// LS Electric XG5000 project: 신호등
// PLC LSPLC

PROGRAM 신호등 (task: 스캔 프로그램)

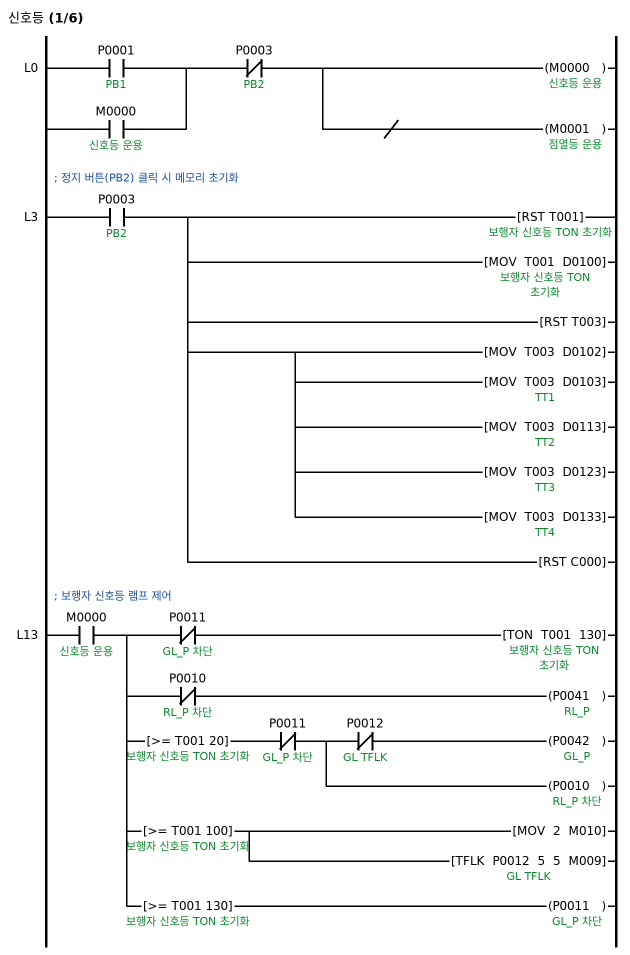
; L0
LOAD      P0001	// PB1
OR        M0000	// 신호등 운용
AND NOT   P0003	// PB2
OUT       M0000	// 신호등 운용
NOT
OUT       M0001	// 점멸등 운용
// 정지 버튼(PB2) 클릭 시 메모리 초기화
; L3
LOAD      P0003	// PB2
RST       T001	// 보행자 신호등 TON 초기화
MOV       T001 D0100	// 보행자 신호등 TON 초기화
RST       T003
MOV       T003 D0102
MOV       T003 D0103	// TT1
MOV       T003 D0113	// TT2
MOV       T003 D0123	// TT3
MOV       T003 D0133	// TT4
RST       C000
// 보행자 신호등 램프 제어
; L13
LOAD      M0000	// 신호등 운용
MPUSH
AND NOT   P0011	// GL_P 차단
TON       T001 130	// 보행자 신호등 TON 초기화
MLOAD
AND NOT   P0010	// RL_P 차단
OUT       P0041	// RL_P
MLOAD
AND>=     T001 20	// 보행자 신호등 TON 초기화
AND NOT   P0011	// GL_P 차단
MPUSH
AND NOT   P0012	// GL TFLK
OUT       P0042	// GL_P
MPOP
OUT       P0010	// RL_P 차단
MLOAD
AND>=     T001 100	// 보행자 신호등 TON 초기화
MOV       2 M010
TFLK      P0012 5 5 M009	// GL TFLK
MPOP
AND>=     T001 130	// 보행자 신호등 TON 초기화
OUT       P0011	// GL_P 차단

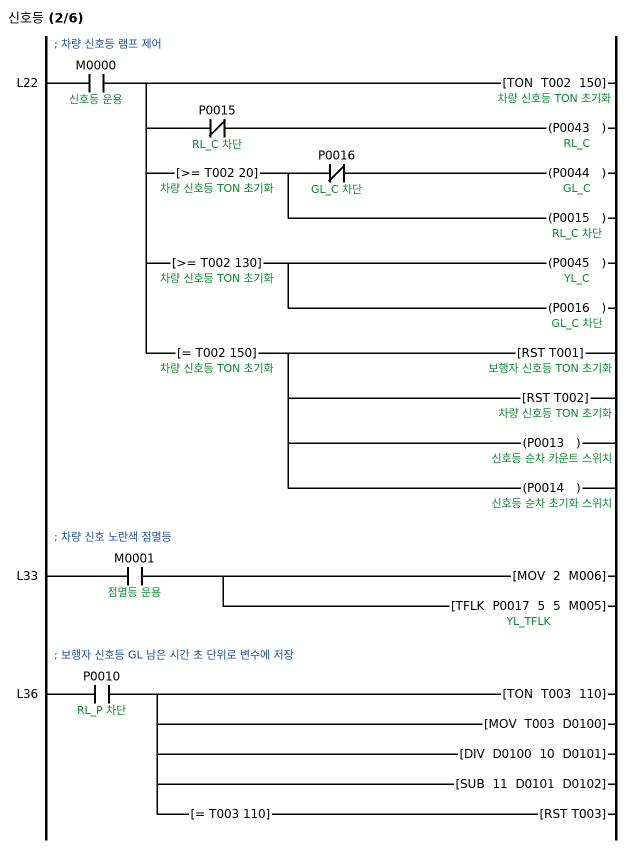
// 차량 신호등 램프 제어
; L22
LOAD      M0000	// 신호등 운용
TON       T002 150	// 차량 신호등 TON 초기화
MPUSH
AND NOT   P0015	// RL_C 차단
OUT       P0043	// RL_C
MLOAD
AND>=     T002 20	// 차량 신호등 TON 초기화
MPUSH
AND NOT   P0016	// GL_C 차단
OUT       P0044	// GL_C
MPOP
OUT       P0015	// RL_C 차단
MLOAD
AND>=     T002 130	// 차량 신호등 TON 초기화
OUT       P0045	// YL_C
OUT       P0016	// GL_C 차단
MPOP
AND=      T002 150	// 차량 신호등 TON 초기화
RST       T001	// 보행자 신호등 TON 초기화
RST       T002	// 차량 신호등 TON 초기화
OUT       P0013	// 신호등 순차 카운트 스위치
OUT       P0014	// 신호등 순차 초기화 스위치
// 차량 신호 노란색 점멸등 
; L33
LOAD      M0001	// 점멸등 운용
MOV       2 M006
TFLK      P0017 5 5 M005	// YL_TFLK
// 보행자 신호등 GL 남은 시간 초 단위로 변수에 저장
; L36
LOAD      P0010	// RL_P 차단
TON       T003 110
MOV       T003 D0100
DIV       D0100 10 D0101
SUB       11 D0101 D0102
AND=      T003 110
RST       T003

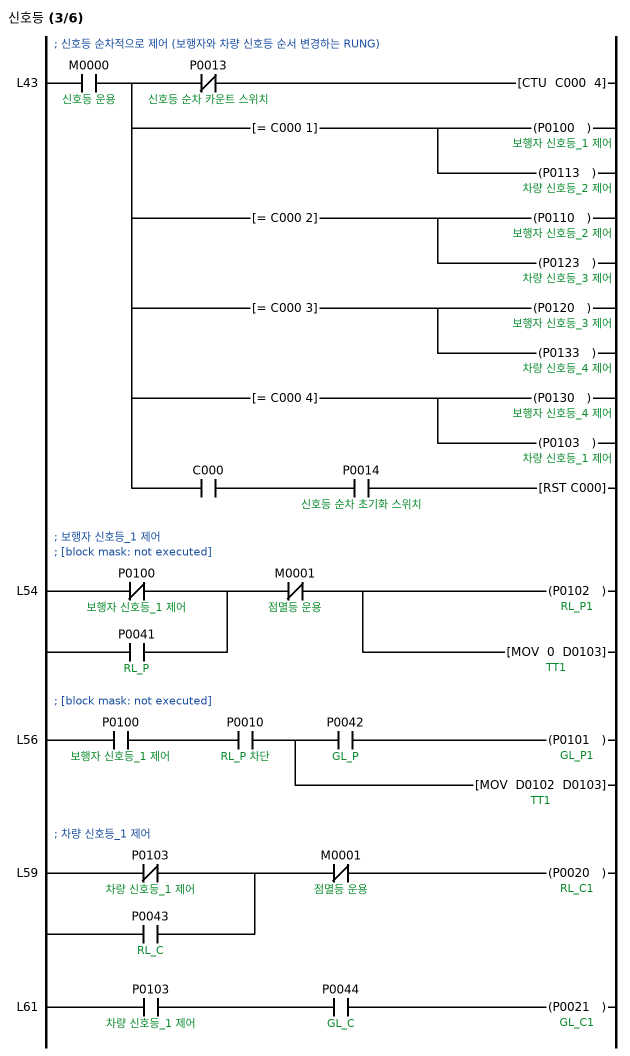
// 신호등 순차적으로 제어 (보행자와 차량 신호등 순서 변경하는 RUNG)
; L43
LOAD      M0000	// 신호등 운용
MPUSH
AND NOT   P0013	// 신호등 순차 카운트 스위치
CTU       C000 4
MLOAD
AND=      C000 1
OUT       P0100	// 보행자 신호등_1 제어
OUT       P0113	// 차량 신호등_2 제어
MLOAD
AND=      C000 2
OUT       P0110	// 보행자 신호등_2 제어
OUT       P0123	// 차량 신호등_3 제어
MLOAD
AND=      C000 3
OUT       P0120	// 보행자 신호등_3 제어
OUT       P0133	// 차량 신호등_4 제어
MLOAD
AND=      C000 4
OUT       P0130	// 보행자 신호등_4 제어
OUT       P0103	// 차량 신호등_1 제어
MPOP
AND       C000
AND       P0014	// 신호등 순차 초기화 스위치
RST       C000
// 보행자 신호등_1 제어
; L54 (block mask: not executed)
LOAD NOT  P0100	// 보행자 신호등_1 제어
OR        P0041	// RL_P
AND NOT   M0001	// 점멸등 운용
OUT       P0102	// RL_P1
MOV       0 D0103	// TT1
; L56 (block mask: not executed)
LOAD      P0100	// 보행자 신호등_1 제어
AND       P0010	// RL_P 차단
MPUSH
AND       P0042	// GL_P
OUT       P0101	// GL_P1
MPOP
MOV       D0102 D0103	// TT1
// 차량 신호등_1 제어
; L59
LOAD NOT  P0103	// 차량 신호등_1 제어
OR        P0043	// RL_C
AND NOT   M0001	// 점멸등 운용
OUT       P0020	// RL_C1
; L61
LOAD      P0103	// 차량 신호등_1 제어
AND       P0044	// GL_C
OUT       P0021	// GL_C1

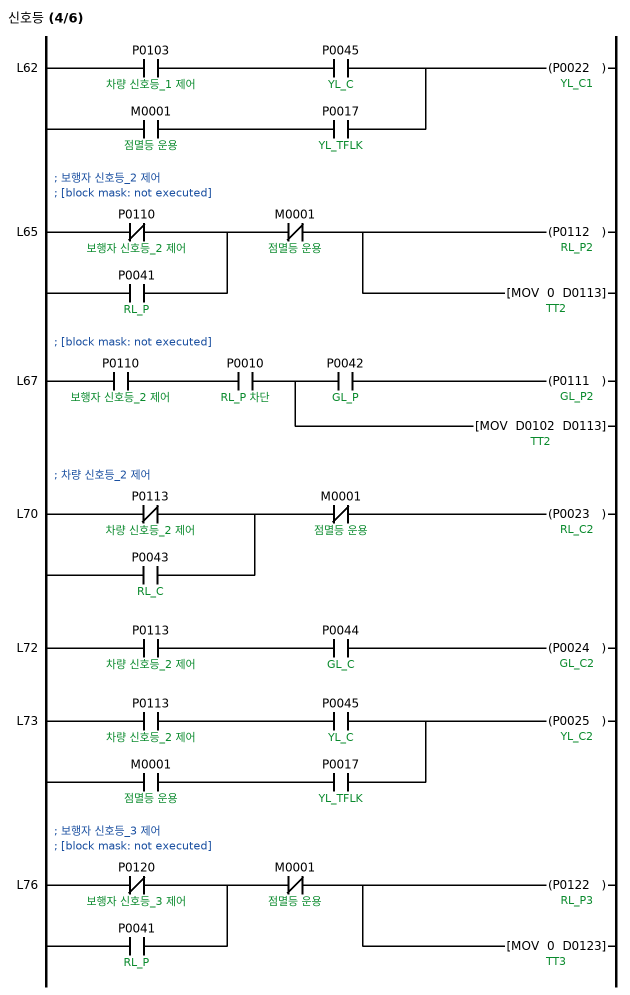
; L62
LOAD      P0103	// 차량 신호등_1 제어
AND       P0045	// YL_C
LOAD      M0001	// 점멸등 운용
AND       P0017	// YL_TFLK
OR LOAD
OUT       P0022	// YL_C1
// 보행자 신호등_2 제어
; L65 (block mask: not executed)
LOAD NOT  P0110	// 보행자 신호등_2 제어
OR        P0041	// RL_P
AND NOT   M0001	// 점멸등 운용
OUT       P0112	// RL_P2
MOV       0 D0113	// TT2
; L67 (block mask: not executed)
LOAD      P0110	// 보행자 신호등_2 제어
AND       P0010	// RL_P 차단
MPUSH
AND       P0042	// GL_P
OUT       P0111	// GL_P2
MPOP
MOV       D0102 D0113	// TT2
// 차량 신호등_2 제어
; L70
LOAD NOT  P0113	// 차량 신호등_2 제어
OR        P0043	// RL_C
AND NOT   M0001	// 점멸등 운용
OUT       P0023	// RL_C2
; L72
LOAD      P0113	// 차량 신호등_2 제어
AND       P0044	// GL_C
OUT       P0024	// GL_C2
; L73
LOAD      P0113	// 차량 신호등_2 제어
AND       P0045	// YL_C
LOAD      M0001	// 점멸등 운용
AND       P0017	// YL_TFLK
OR LOAD
OUT       P0025	// YL_C2
// 보행자 신호등_3 제어
; L76 (block mask: not executed)
LOAD NOT  P0120	// 보행자 신호등_3 제어
OR        P0041	// RL_P
AND NOT   M0001	// 점멸등 운용
OUT       P0122	// RL_P3
MOV       0 D0123	// TT3

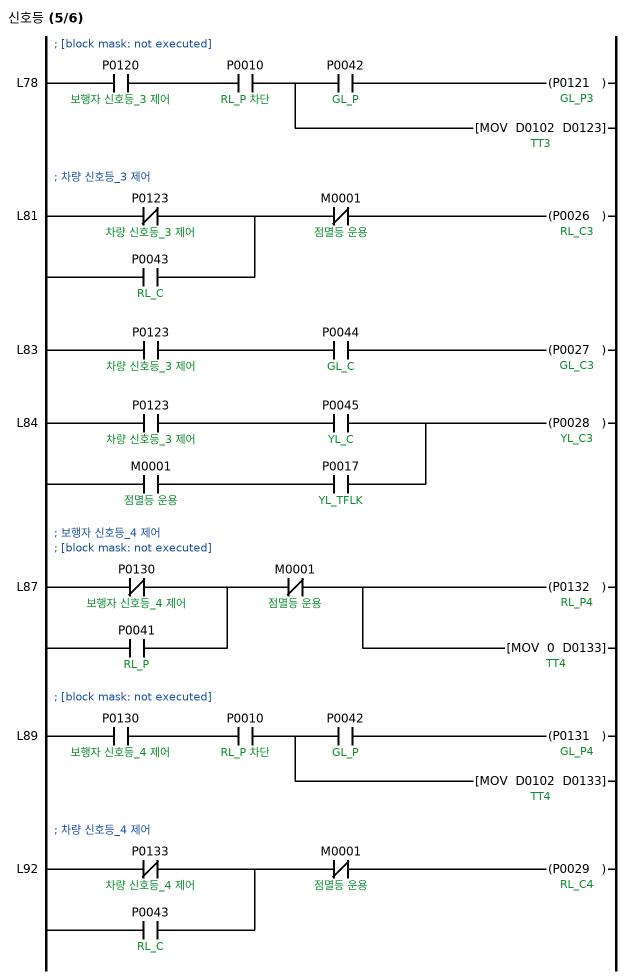
; L78 (block mask: not executed)
LOAD      P0120	// 보행자 신호등_3 제어
AND       P0010	// RL_P 차단
MPUSH
AND       P0042	// GL_P
OUT       P0121	// GL_P3
MPOP
MOV       D0102 D0123	// TT3
// 차량 신호등_3 제어
; L81
LOAD NOT  P0123	// 차량 신호등_3 제어
OR        P0043	// RL_C
AND NOT   M0001	// 점멸등 운용
OUT       P0026	// RL_C3
; L83
LOAD      P0123	// 차량 신호등_3 제어
AND       P0044	// GL_C
OUT       P0027	// GL_C3
; L84
LOAD      P0123	// 차량 신호등_3 제어
AND       P0045	// YL_C
LOAD      M0001	// 점멸등 운용
AND       P0017	// YL_TFLK
OR LOAD
OUT       P0028	// YL_C3
// 보행자 신호등_4 제어
; L87 (block mask: not executed)
LOAD NOT  P0130	// 보행자 신호등_4 제어
OR        P0041	// RL_P
AND NOT   M0001	// 점멸등 운용
OUT       P0132	// RL_P4
MOV       0 D0133	// TT4
; L89 (block mask: not executed)
LOAD      P0130	// 보행자 신호등_4 제어
AND       P0010	// RL_P 차단
MPUSH
AND       P0042	// GL_P
OUT       P0131	// GL_P4
MPOP
MOV       D0102 D0133	// TT4
// 차량 신호등_4 제어
; L92
LOAD NOT  P0133	// 차량 신호등_4 제어
OR        P0043	// RL_C
AND NOT   M0001	// 점멸등 운용
OUT       P0029	// RL_C4

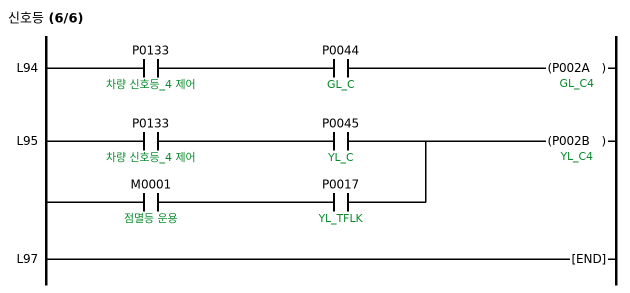
; L94
LOAD      P0133	// 차량 신호등_4 제어
AND       P0044	// GL_C
OUT       P002A	// GL_C4
; L95
LOAD      P0133	// 차량 신호등_4 제어
AND       P0045	// YL_C
LOAD      M0001	// 점멸등 운용
AND       P0017	// YL_TFLK
OR LOAD
OUT       P002B	// YL_C4
; L97
END

VARIABLES AND COMMENTS (devices not used above)
P00004	BIT	PB4